Universal Robots PolyScope program: tower.urp

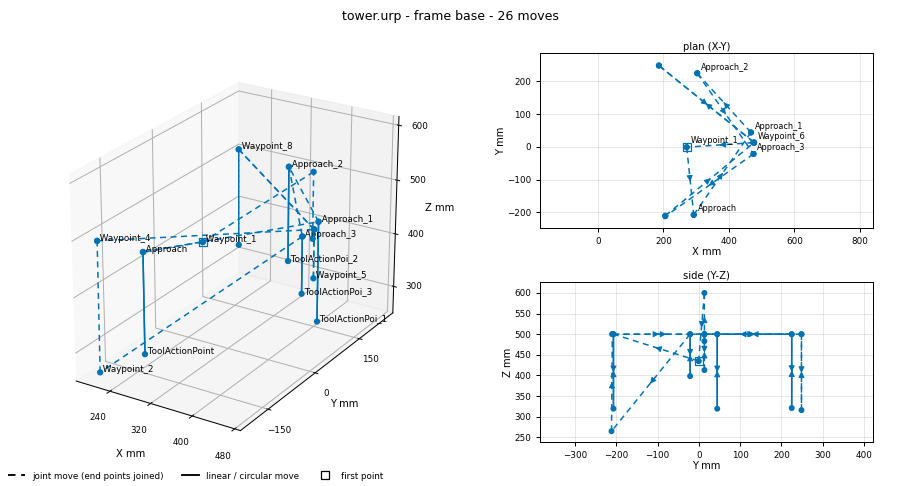
[picture p0: tool path of tower.urp in frame base, 26 of 26 moves have a stored position in this frame; points joined in program order, loops and branches not executed]
Program tower (installation=default directory=/programs createdIn=5.11.9.1010452 lastSavedIn=5.11.9.1010452 robotSerialNumber=20225200364)
Calibrated DH parameters: a=[0.00002, -0.569483, -0.54992, -0.00001, -0.000036, 0]; d=[0.180894, -146.691669, 192.918669, -46.053088, 0.119778, 0.115602]; alpha=[1.571425, -0.001534, 0.003359, 1.568739, -1.571477, 0]; deltaTheta=[0, 0.376258, -0.101074, -0.275185, -0.000002, 0]
Robot Program (runOnlyOnce=false)
  URCap RG Grip (OnRobot, OnRobot A/S) dataModel(rg-target-force=40.0, rg-target-width=0.1, Variable(key=on_return, variable(name=on_return)))
  MoveJ speed 60 deg/s, acceleration 80 deg/s^2 (useActiveTCP=true) feature=Base
    Waypoint Waypoint_1: TCP in base x=271.114 y=-0.718 z=434.853 mm, rx=2.1943 ry=2.2475 rz=0.0032 rad; joints [39.865, -70.399, -130.922, 111.401, -90.192, 38.695] deg
    Loop Counting (count=3) loopVariable(name=Loop_1)
      URCap Palletizing (polyscope-pallet-impl, Universal Robots) dataModel(palletFeature=Base, isPalletizing=true, Variable(key=name, variable(name=Pallet_1)), Variable(key=globalCountingVariable, variable(name=Pallet_1_cnt_1, initializeExpression=1)), Variable(key=layerNumberVariable, variable(name=Pallet_1_lno, initializeExpression=1)), Variable(key=layerCountingVariable, variable(name=Pallet_1_lct, initializeExpression=1)), Variable(key=handleSeparatorVariable, variable(name=Pallet_1_sep, initializeExpression=False)), Variable(key=totalCountVariable, variable(name=Pallet_1_tct, initializeExpression=1)), Variable(key=referencePoint, variable(featureName=referencePoint)), Variable(key=separatorPoint, variable(featureName=separatorPoint)), Length(key=objectHeight value=0.00001 unit=M)); state(isChildrenLocked=true)
        URCap Patterns (polyscope-pallet-impl, Universal Robots) state(isChildrenLocked=true)
          URCap Pattern (polyscope-pallet-impl, Universal Robots) dataModel(UUID=10b702ad-919e-447e-83f3-c5d126601516, patternType=LINE, objects=3, Variable(key=nameVariable, variable(name=Line_Pattern_1))); state(isChildrenLocked=true)
            URCap Item (polyscope-pallet-impl, Universal Robots) dataModel(UUID=ffec0e32-995c-4917-bab5-c4ad35439001, patternType=LINE, index=0, calibrationDeltaTheta=[-2.1094217540068572E-7, 0.37625772532806073, -0.10107441100396769, -0.2751850025766889, -1.8024952768980196E-6, 2.9402326063437956E-8], calibrationA=[2.0416891277915125E-5, -0.5694828868469309, -0.5499202125525207, -9.504674691390763E-6, -3.603723657207661E-5, 0.0], calibrationD=[0.1808937726775539, -146.69166934821124, 192.91866861971778, -46.05308757405963, 0.11977780403821288, 0.11560212559305974], calibrationAlpha=[1.5714252480212174, -0.0015337665762078037, 0.0033588312559612306, 1.5687392298942362, -1.5714772428732047, 0.0], calibrationJointChecksum=[-1490546360, -1456574554, -1506622700, -1493399207, -1492840923, -1492940558], calibrationStatus=2, calibrationValidChecksum=true, baseToFeature=[0.0, 0.0, 0.0, 0.0, 0.0, 0.0], TCPOffset=[-6.3696764394660654E-6, 1.3718254129935215E-5, 1.7975052069185704E-5, -3.893490764890671E-5, -1.8800917890220025E-5, -2.364729783574531E-6], Variable(key=variable, variable(name=StartItem_1)), JointPositions(key=jointpositions, JointPosition(key=[1], Angle(key=pos value=-0.12044 unit=RAD)), JointPosition(key=[2], Angle(key=pos value=-1.547684 unit=RAD)), JointPosition(key=[3], Angle(key=pos value=-2.267587 unit=RAD)), JointPosition(key=[4], Angle(key=pos value=2.262922 unit=RAD)), JointPosition(key=[5], Angle(key=pos value=-1.606027 unit=RAD)), JointPosition(key=[6], Angle(key=pos value=2.964753 unit=RAD))))
            URCap Item (polyscope-pallet-impl, Universal Robots) dataModel(UUID=13b54a3e-8037-4e83-825c-96e2be57fcbd, patternType=LINE, index=1, calibrationDeltaTheta=[-2.1094217540068572E-7, 0.37625772532806073, -0.10107441100396769, -0.2751850025766889, -1.8024952768980196E-6, 2.9402326063437956E-8], calibrationA=[2.0416891277915125E-5, -0.5694828868469309, -0.5499202125525207, -9.504674691390763E-6, -3.603723657207661E-5, 0.0], calibrationD=[0.1808937726775539, -146.69166934821124, 192.91866861971778, -46.05308757405963, 0.11977780403821288, 0.11560212559305974], calibrationAlpha=[1.5714252480212174, -0.0015337665762078037, 0.0033588312559612306, 1.5687392298942362, -1.5714772428732047, 0.0], calibrationJointChecksum=[-1490546360, -1456574554, -1506622700, -1493399207, -1492840923, -1492940558], calibrationStatus=2, calibrationValidChecksum=true, baseToFeature=[0.0, 0.0, 0.0, 0.0, 0.0, 0.0], TCPOffset=[1.3846566568914698E-5, -1.1531112679291633E-5, -9.126227575095847E-6, 3.8309900976807E-6, 1.563735032861701E-5, 6.604035696750426E-5], Variable(key=variable, variable(name=EndItem_1)), JointPositions(key=jointpositions, JointPosition(key=[1], Angle(key=pos value=-0.160653 unit=RAD)), JointPosition(key=[2], Angle(key=pos value=-1.420785 unit=RAD)), JointPosition(key=[3], Angle(key=pos value=-2.379964 unit=RAD)), JointPosition(key=[4], Angle(key=pos value=2.247089 unit=RAD)), JointPosition(key=[5], Angle(key=pos value=-1.606961 unit=RAD)), JointPosition(key=[6], Angle(key=pos value=2.924393 unit=RAD))))
        URCap Layers (polyscope-pallet-impl, Universal Robots) dataModel(separators=[false], selectedPatterns=[10b702ad-919e-447e-83f3-c5d126601516])
        URCap At Each Item (polyscope-pallet-impl, Universal Robots) dataModel(selectedPattern=10b702ad-919e-447e-83f3-c5d126601516, selectedPosition=ffec0e32-995c-4917-bab5-c4ad35439001, Approach_calibrationDeltaTheta=[-2.1094217540068572E-7, 0.37625772532806073, -0.10107441100396769, -0.2751850025766889, -1.8024952768980196E-6, 2.9402326063437956E-8], Approach_calibrationA=[2.0416891277915125E-5, -0.5694828868469309, -0.5499202125525207, -9.504674691390763E-6, -3.603723657207661E-5, 0.0], Approach_calibrationD=[0.1808937726775539, -146.69166934821124, 192.91866861971778, -46.05308757405963, 0.11977780403821288, 0.11560212559305974], Approach_calibrationAlpha=[1.5714252480212174, -0.0015337665762078037, 0.0033588312559612306, 1.5687392298942362, -1.5714772428732047, 0.0], Approach_calibrationJointChecksum=[-1490546360, -1456574554, -1506622700, -1493399207, -1492840923, -1492940558], Approach_calibrationStatus=2, Approach_calibrationValidChecksum=true, Approach_baseToFeature=[0.0, 0.0, 0.0, 0.0, 0.0, 0.0], Approach_TCPOffset=[4.62405650436537E-8, -1.550057465476984E-5, -1.2608941560687814E-5, -1.6491377497452102E-5, -2.0027642314724937E-5, -1.4317350537033054E-5], Exit_calibrationDeltaTheta=[-2.1094217540068572E-7, 0.37625772532806073, -0.10107441100396769, -0.2751850025766889, -1.8024952768980196E-6, 2.9402326063437956E-8], Exit_calibrationA=[2.0416891277915125E-5, -0.5694828868469309, -0.5499202125525207, -9.504674691390763E-6, -3.603723657207661E-5, 0.0], Exit_calibrationD=[0.1808937726775539, -146.69166934821124, 192.91866861971778, -46.05308757405963, 0.11977780403821288, 0.11560212559305974], Exit_calibrationAlpha=[1.5714252480212174, -0.0015337665762078037, 0.0033588312559612306, 1.5687392298942362, -1.5714772428732047, 0.0], Exit_calibrationJointChecksum=[-1490546360, -1456574554, -1506622700, -1493399207, -1492840923, -1492940558], Exit_calibrationStatus=2, Exit_calibrationValidChecksum=true, Exit_baseToFeature=[0.0, 0.0, 0.0, 0.0, 0.0, 0.0], Exit_TCPOffset=[1.1446723165831063E-5, 3.368334611741908E-5, -1.8687979546572198E-5, 3.7324910344696995E-5, 7.929792478961527E-6, 6.655834368709218E-5], currentWizardState=LANDING, Pose(key=refBaseToFeature, Position(key=posePosition, Length(key=X value=0 unit=M), Length(key=Y value=0 unit=M), Length(key=Z value=0 unit=M)), Rotation(key=poseRotation, Angle(key=RX value=0 unit=RAD), Angle(key=RY value=0 unit=RAD), Angle(key=RZ value=0 unit=RAD))), Pose(key=refPose, Position(key=posePosition, Length(key=X value=0.29256 unit=M), Length(key=Y value=-0.207279 unit=M), Length(key=Z value=0.319351 unit=M)), Rotation(key=poseRotation, Angle(key=RX value=-2.261622 unit=RAD), Angle(key=RY value=2.126603 unit=RAD), Angle(key=RZ value=0.005998 unit=RAD))), JointPositions(key=Approach_jointpositions, JointPosition(key=[1], Angle(key=pos value=-0.121062 unit=RAD)), JointPosition(key=[2], Angle(key=pos value=-1.383215 unit=RAD)), JointPosition(key=[3], Angle(key=pos value=-2.051976 unit=RAD)), JointPosition(key=[4], Angle(key=pos value=1.882818 unit=RAD)), JointPosition(key=[5], Angle(key=pos value=-1.606548 unit=RAD)), JointPosition(key=[6], Angle(key=pos value=2.962745 unit=RAD))), JointPositions(key=Exit_jointpositions, JointPosition(key=[1], Angle(key=pos value=-0.121058 unit=RAD)), JointPosition(key=[2], Angle(key=pos value=-1.383222 unit=RAD)), JointPosition(key=[3], Angle(key=pos value=-2.051981 unit=RAD)), JointPosition(key=[4], Angle(key=pos value=1.88278 unit=RAD)), JointPosition(key=[5], Angle(key=pos value=-1.606525 unit=RAD)), JointPosition(key=[6], Angle(key=pos value=2.962785 unit=RAD))))
          URCap Generated Movements (polyscope-pallet-impl, Universal Robots) state(isChildrenLocked=true)
            MoveJ speed 60 deg/s, acceleration 80 deg/s^2 (useActiveTCP=true) feature=referencePoint
              Waypoint Approach: TCP in base x=292.598 y=-207.278 z=500.013 mm, rx=-2.2616 ry=2.1265 rz=0.0059 rad; joints [-6.936, -79.254, -117.567, 107.876, -92.049, 169.752] deg; TCP offset x=0 y=0 z=0 mm, rx=0 ry=0 rz=0 rad; feature pose in base x=292.56 y=-207.279 z=319.351 mm, rx=-2.2616 ry=2.1266 rz=0.006 rad
            MoveL speed 250 mm/s, acceleration 1200 mm/s^2 (useActiveTCP=true) feature(featureName=referencePoint)
              Waypoint ToolActionPoint: TCP in base x=292.56 y=-207.279 z=319.351 mm, rx=-2.2616 ry=2.1266 rz=0.006 rad; joints [-6.9, -88.676, -129.925, 129.656, -92.019, 169.868] deg; TCP offset x=0 y=0 z=0 mm, rx=0 ry=0 rz=0 rad
            Folder Tool action
              URCap RG Grip (OnRobot, OnRobot A/S) dataModel(rg-target-force=40.0, rg-target-width=0.025)
            MoveL speed 250 mm/s, acceleration 1200 mm/s^2 (useActiveTCP=true) feature(featureName=referencePoint)
              Waypoint Exit_1: TCP in base x=292.546 y=-207.293 z=500.018 mm, rx=-2.2615 ry=2.1267 rz=0.0059 rad; joints [-6.939, -79.249, -117.57, 107.874, -92.047, 169.756] deg; TCP offset x=0 y=0 z=0 mm, rx=0 ry=0 rz=0 rad
      URCap Palletizing (polyscope-pallet-impl, Universal Robots) dataModel(palletFeature=Base, isPalletizing=true, Variable(key=name, variable(name=Pallet_2)), Variable(key=globalCountingVariable, variable(name=Pallet_2_cnt, initializeExpression=1)), Variable(key=layerNumberVariable, variable(name=Pallet_2_lno, initializeExpression=1)), Variable(key=layerCountingVariable, variable(name=Pallet_2_lct, initializeExpression=1)), Variable(key=handleSeparatorVariable, variable(name=Pallet_2_sep, initializeExpression=False)), Variable(key=totalCountVariable, variable(name=Pallet_2_tct, initializeExpression=1)), Variable(key=referencePoint, variable(featureName=referencePoin_1)), Variable(key=separatorPoint, variable(featureName=separatorPoin_1)), Length(key=objectHeight value=0.00001 unit=M)); state(isChildrenLocked=true)
        URCap Patterns (polyscope-pallet-impl, Universal Robots) state(isChildrenLocked=true)
          URCap Pattern (polyscope-pallet-impl, Universal Robots) dataModel(UUID=c8f087d8-a87e-4c62-a9c1-169a6018fd4e, patternType=LINE, objects=3, Variable(key=nameVariable, variable(name=Line_Pattern_2))); state(isChildrenLocked=true)
            URCap Item (polyscope-pallet-impl, Universal Robots) dataModel(UUID=4b9336ee-f1af-4d45-8009-66d60779b6a6, patternType=LINE, index=0, calibrationDeltaTheta=[-2.1094217540068572E-7, 0.37625772532806073, -0.10107441100396769, -0.2751850025766889, -1.8024952768980196E-6, 2.9402326063437956E-8], calibrationA=[2.0416891277915125E-5, -0.5694828868469309, -0.5499202125525207, -9.504674691390763E-6, -3.603723657207661E-5, 0.0], calibrationD=[0.1808937726775539, -146.69166934821124, 192.91866861971778, -46.05308757405963, 0.11977780403821288, 0.11560212559305974], calibrationAlpha=[1.5714252480212174, -0.0015337665762078037, 0.0033588312559612306, 1.5687392298942362, -1.5714772428732047, 0.0], calibrationJointChecksum=[-1490546360, -1456574554, -1506622700, -1493399207, -1492840923, -1492940558], calibrationStatus=2, calibrationValidChecksum=true, baseToFeature=[0.0, 0.0, 0.0, 0.0, 0.0, 0.0], TCPOffset=[4.409116630077481E-6, -1.5438319090163577E-5, -7.2719913739582864E-6, 5.112219757212625E-5, -6.20493439311258E-5, 5.425001136176107E-5], Variable(key=variable, variable(name=StartItem_2)), JointPositions(key=jointpositions, JointPosition(key=[1], Angle(key=pos value=0.474651 unit=RAD)), JointPosition(key=[2], Angle(key=pos value=-1.730821 unit=RAD)), JointPosition(key=[3], Angle(key=pos value=-2.064013 unit=RAD)), JointPosition(key=[4], Angle(key=pos value=2.256065 unit=RAD)), JointPosition(key=[5], Angle(key=pos value=-1.574508 unit=RAD)), JointPosition(key=[6], Angle(key=pos value=5.17627 unit=RAD))))
            URCap Item (polyscope-pallet-impl, Universal Robots) dataModel(UUID=a110d0e4-b9f2-4c4c-afd7-8c47bd34fb09, patternType=LINE, index=1, calibrationDeltaTheta=[-2.1094217540068572E-7, 0.37625772532806073, -0.10107441100396769, -0.2751850025766889, -1.8024952768980196E-6, 2.9402326063437956E-8], calibrationA=[2.0416891277915125E-5, -0.5694828868469309, -0.5499202125525207, -9.504674691390763E-6, -3.603723657207661E-5, 0.0], calibrationD=[0.1808937726775539, -146.69166934821124, 192.91866861971778, -46.05308757405963, 0.11977780403821288, 0.11560212559305974], calibrationAlpha=[1.5714252480212174, -0.0015337665762078037, 0.0033588312559612306, 1.5687392298942362, -1.5714772428732047, 0.0], calibrationJointChecksum=[-1490546360, -1456574554, -1506622700, -1493399207, -1492840923, -1492940558], calibrationStatus=2, calibrationValidChecksum=true, baseToFeature=[0.0, 0.0, 0.0, 0.0, 0.0, 0.0], TCPOffset=[-1.4380333733965411E-5, -5.264472437292028E-6, -9.358425566097228E-6, -1.0911522351191877E-5, -4.3963888238967464E-5, 2.2254276518748705E-5], Variable(key=variable, variable(name=EndItem_2)), JointPositions(key=jointpositions, JointPosition(key=[1], Angle(key=pos value=0.326248 unit=RAD)), JointPosition(key=[2], Angle(key=pos value=-1.729038 unit=RAD)), JointPosition(key=[3], Angle(key=pos value=-2.066304 unit=RAD)), JointPosition(key=[4], Angle(key=pos value=2.256092 unit=RAD)), JointPosition(key=[5], Angle(key=pos value=-1.579334 unit=RAD)), JointPosition(key=[6], Angle(key=pos value=5.027941 unit=RAD))))
        URCap Layers (polyscope-pallet-impl, Universal Robots) dataModel(separators=[false], selectedPatterns=[c8f087d8-a87e-4c62-a9c1-169a6018fd4e])
        URCap At Each Item (polyscope-pallet-impl, Universal Robots) dataModel(selectedPattern=c8f087d8-a87e-4c62-a9c1-169a6018fd4e, selectedPosition=4b9336ee-f1af-4d45-8009-66d60779b6a6, Approach_calibrationDeltaTheta=[-2.1094217540068572E-7, 0.37625772532806073, -0.10107441100396769, -0.2751850025766889, -1.8024952768980196E-6, 2.9402326063437956E-8], Approach_calibrationA=[2.0416891277915125E-5, -0.5694828868469309, -0.5499202125525207, -9.504674691390763E-6, -3.603723657207661E-5, 0.0], Approach_calibrationD=[0.1808937726775539, -146.69166934821124, 192.91866861971778, -46.05308757405963, 0.11977780403821288, 0.11560212559305974], Approach_calibrationAlpha=[1.5714252480212174, -0.0015337665762078037, 0.0033588312559612306, 1.5687392298942362, -1.5714772428732047, 0.0], Approach_calibrationJointChecksum=[-1490546360, -1456574554, -1506622700, -1493399207, -1492840923, -1492940558], Approach_calibrationStatus=2, Approach_calibrationValidChecksum=true, Approach_baseToFeature=[0.0, 0.0, 0.0, 0.0, 0.0, 0.0], Approach_TCPOffset=[1.1639698013432564E-5, -8.846874539378269E-6, 1.1133412487873695E-5, 1.6117839583191827E-5, 5.374636367245953E-5, 1.074239401068827E-6], Exit_calibrationDeltaTheta=[-2.1094217540068572E-7, 0.37625772532806073, -0.10107441100396769, -0.2751850025766889, -1.8024952768980196E-6, 2.9402326063437956E-8], Exit_calibrationA=[2.0416891277915125E-5, -0.5694828868469309, -0.5499202125525207, -9.504674691390763E-6, -3.603723657207661E-5, 0.0], Exit_calibrationD=[0.1808937726775539, -146.69166934821124, 192.91866861971778, -46.05308757405963, 0.11977780403821288, 0.11560212559305974], Exit_calibrationAlpha=[1.5714252480212174, -0.0015337665762078037, 0.0033588312559612306, 1.5687392298942362, -1.5714772428732047, 0.0], Exit_calibrationJointChecksum=[-1490546360, -1456574554, -1506622700, -1493399207, -1492840923, -1492940558], Exit_calibrationStatus=2, Exit_calibrationValidChecksum=true, Exit_baseToFeature=[0.0, 0.0, 0.0, 0.0, 0.0, 0.0], Exit_TCPOffset=[-6.688063342030759E-8, 1.0405827377074628E-5, -5.466452467406402E-6, 3.1866222240658605E-5, 4.424926447771402E-5, -4.5818155317012656E-5], currentWizardState=LANDING, Pose(key=refBaseToFeature, Position(key=posePosition, Length(key=X value=0 unit=M), Length(key=Y value=0 unit=M), Length(key=Z value=0 unit=M)), Rotation(key=poseRotation, Angle(key=RX value=0 unit=RAD), Angle(key=RY value=0 unit=RAD), Angle(key=RZ value=0 unit=RAD))), Pose(key=refPose, Position(key=posePosition, Length(key=X value=0.46728 unit=M), Length(key=Y value=0.044349 unit=M), Length(key=Z value=0.319231 unit=M)), Rotation(key=poseRotation, Angle(key=RX value=-0.0243 unit=RAD), Angle(key=RY value=3.112588 unit=RAD), Angle(key=RZ value=0.024192 unit=RAD))), JointPositions(key=Approach_jointpositions, JointPosition(key=[1], Angle(key=pos value=0.474285 unit=RAD)), JointPosition(key=[2], Angle(key=pos value=-1.582914 unit=RAD)), JointPosition(key=[3], Angle(key=pos value=-1.86876 unit=RAD)), JointPosition(key=[4], Angle(key=pos value=1.91298 unit=RAD)), JointPosition(key=[5], Angle(key=pos value=-1.574975 unit=RAD)), JointPosition(key=[6], Angle(key=pos value=5.174807 unit=RAD))), JointPositions(key=Exit_jointpositions, JointPosition(key=[1], Angle(key=pos value=0.474302 unit=RAD)), JointPosition(key=[2], Angle(key=pos value=-1.582917 unit=RAD)), JointPosition(key=[3], Angle(key=pos value=-1.868746 unit=RAD)), JointPosition(key=[4], Angle(key=pos value=1.913021 unit=RAD)), JointPosition(key=[5], Angle(key=pos value=-1.574942 unit=RAD)), JointPosition(key=[6], Angle(key=pos value=5.174836 unit=RAD))))
          URCap Generated Movements (polyscope-pallet-impl, Universal Robots) state(isChildrenLocked=true)
            MoveJ speed 60 deg/s, acceleration 80 deg/s^2 (useActiveTCP=true) feature=referencePoin_1
              Waypoint Approach_1: TCP in base x=467.265 y=44.333 z=499.988 mm, rx=-0.0243 ry=3.1126 rz=0.0243 rad; joints [27.174, -90.694, -107.074, 109.604, -90.24, 296.494] deg; TCP offset x=0 y=0 z=0 mm, rx=0 ry=0 rz=0 rad; feature pose in base x=467.28 y=44.349 z=319.231 mm, rx=-0.0243 ry=3.1126 rz=0.0242 rad
            MoveL speed 250 mm/s, acceleration 1200 mm/s^2 (useActiveTCP=true) feature(featureName=referencePoin_1)
              Waypoint ToolActionPoi_1: TCP in base x=467.28 y=44.349 z=319.231 mm, rx=-0.0243 ry=3.1126 rz=0.0242 rad; joints [27.195, -99.167, -118.26, 129.264, -90.208, 296.581] deg; TCP offset x=0 y=0 z=0 mm, rx=0 ry=0 rz=0 rad
            Folder Tool action
              URCap RG Grip (OnRobot, OnRobot A/S) dataModel(rg-target-force=40.0, rg-target-width=0.03)
            MoveL speed 250 mm/s, acceleration 1200 mm/s^2 (useActiveTCP=true) feature(featureName=referencePoin_1)
              Waypoint Exit_2: TCP in base x=467.286 y=44.361 z=500.006 mm, rx=-0.0243 ry=3.1125 rz=0.0242 rad; joints [27.177, -90.695, -107.071, 109.605, -90.237, 296.495] deg; TCP offset x=0 y=0 z=0 mm, rx=0 ry=0 rz=0 rad
    Loop Counting (count=3) loopVariable(name=Loop_2)
      URCap Palletizing (polyscope-pallet-impl, Universal Robots) dataModel(palletFeature=Base, isPalletizing=true, Variable(key=name, variable(name=Pallet_3)), Variable(key=globalCountingVariable, variable(name=Pallet_3_cnt, initializeExpression=1)), Variable(key=layerNumberVariable, variable(name=Pallet_3_lno, initializeExpression=1)), Variable(key=layerCountingVariable, variable(name=Pallet_3_lct, initializeExpression=1)), Variable(key=handleSeparatorVariable, variable(name=Pallet_3_sep, initializeExpression=False)), Variable(key=totalCountVariable, variable(name=Pallet_3_tct, initializeExpression=1)), Variable(key=referencePoint, variable(featureName=referencePoin_2)), Variable(key=separatorPoint, variable(featureName=separatorPoin_2)), Length(key=objectHeight value=0.00001 unit=M)); state(isChildrenLocked=true)
        URCap Patterns (polyscope-pallet-impl, Universal Robots) state(isChildrenLocked=true)
          URCap Pattern (polyscope-pallet-impl, Universal Robots) dataModel(UUID=69e63fbd-ac57-40a8-8514-40e488ea7127, patternType=LINE, objects=3, Variable(key=nameVariable, variable(name=Line_Pattern_3))); state(isChildrenLocked=true)
            URCap Item (polyscope-pallet-impl, Universal Robots) dataModel(UUID=d74f1e55-d7a4-4b92-9c14-17e5686717f3, patternType=LINE, index=0, calibrationDeltaTheta=[-2.1094217540068572E-7, 0.37625772532806073, -0.10107441100396769, -0.2751850025766889, -1.8024952768980196E-6, 2.9402326063437956E-8], calibrationA=[2.0416891277915125E-5, -0.5694828868469309, -0.5499202125525207, -9.504674691390763E-6, -3.603723657207661E-5, 0.0], calibrationD=[0.1808937726775539, -146.69166934821124, 192.91866861971778, -46.05308757405963, 0.11977780403821288, 0.11560212559305974], calibrationAlpha=[1.5714252480212174, -0.0015337665762078037, 0.0033588312559612306, 1.5687392298942362, -1.5714772428732047, 0.0], calibrationJointChecksum=[-1490546360, -1456574554, -1506622700, -1493399207, -1492840923, -1492940558], calibrationStatus=2, calibrationValidChecksum=true, baseToFeature=[0.0, 0.0, 0.0, 0.0, 0.0, 0.0], TCPOffset=[1.2985872193088666E-5, -6.705328385370191E-6, -7.116337871981848E-6, 1.0691414030932002E-5, -1.1363978627081674E-5, -2.520531805839135E-5], Variable(key=variable, variable(name=StartItem_3)), JointPositions(key=jointpositions, JointPosition(key=[1], Angle(key=pos value=1.118695 unit=RAD)), JointPosition(key=[2], Angle(key=pos value=-1.583327 unit=RAD)), JointPosition(key=[3], Angle(key=pos value=-2.233039 unit=RAD)), JointPosition(key=[4], Angle(key=pos value=2.246663 unit=RAD)), JointPosition(key=[5], Angle(key=pos value=-1.572601 unit=RAD)), JointPosition(key=[6], Angle(key=pos value=1.099535 unit=RAD))))
            URCap Item (polyscope-pallet-impl, Universal Robots) dataModel(UUID=ef41c16a-ce02-4892-a50c-4f21fb1603f3, patternType=LINE, index=1, calibrationDeltaTheta=[-2.1094217540068572E-7, 0.37625772532806073, -0.10107441100396769, -0.2751850025766889, -1.8024952768980196E-6, 2.9402326063437956E-8], calibrationA=[2.0416891277915125E-5, -0.5694828868469309, -0.5499202125525207, -9.504674691390763E-6, -3.603723657207661E-5, 0.0], calibrationD=[0.1808937726775539, -146.69166934821124, 192.91866861971778, -46.05308757405963, 0.11977780403821288, 0.11560212559305974], calibrationAlpha=[1.5714252480212174, -0.0015337665762078037, 0.0033588312559612306, 1.5687392298942362, -1.5714772428732047, 0.0], calibrationJointChecksum=[-1490546360, -1456574554, -1506622700, -1493399207, -1492840923, -1492940558], calibrationStatus=2, calibrationValidChecksum=true, baseToFeature=[0.0, 0.0, 0.0, 0.0, 0.0, 0.0], TCPOffset=[-5.307224317796511E-7, -5.42229024316776E-6, -2.5424014468145018E-6, -2.8661002424582808E-5, -9.543783619449082E-6, -3.3871828536279686E-5], Variable(key=variable, variable(name=EndItem_3)), JointPositions(key=jointpositions, JointPosition(key=[1], Angle(key=pos value=1.374483 unit=RAD)), JointPosition(key=[2], Angle(key=pos value=-1.463304 unit=RAD)), JointPosition(key=[3], Angle(key=pos value=-2.345439 unit=RAD)), JointPosition(key=[4], Angle(key=pos value=2.238646 unit=RAD)), JointPosition(key=[5], Angle(key=pos value=-1.572398 unit=RAD)), JointPosition(key=[6], Angle(key=pos value=1.355219 unit=RAD))))
        URCap Layers (polyscope-pallet-impl, Universal Robots) dataModel(separators=[false], selectedPatterns=[69e63fbd-ac57-40a8-8514-40e488ea7127])
        URCap At Each Item (polyscope-pallet-impl, Universal Robots) dataModel(selectedPattern=69e63fbd-ac57-40a8-8514-40e488ea7127, selectedPosition=d74f1e55-d7a4-4b92-9c14-17e5686717f3, Approach_calibrationDeltaTheta=[-2.1094217540068572E-7, 0.37625772532806073, -0.10107441100396769, -0.2751850025766889, -1.8024952768980196E-6, 2.9402326063437956E-8], Approach_calibrationA=[2.0416891277915125E-5, -0.5694828868469309, -0.5499202125525207, -9.504674691390763E-6, -3.603723657207661E-5, 0.0], Approach_calibrationD=[0.1808937726775539, -146.69166934821124, 192.91866861971778, -46.05308757405963, 0.11977780403821288, 0.11560212559305974], Approach_calibrationAlpha=[1.5714252480212174, -0.0015337665762078037, 0.0033588312559612306, 1.5687392298942362, -1.5714772428732047, 0.0], Approach_calibrationJointChecksum=[-1490546360, -1456574554, -1506622700, -1493399207, -1492840923, -1492940558], Approach_calibrationStatus=2, Approach_calibrationValidChecksum=true, Approach_baseToFeature=[0.0, 0.0, 0.0, 0.0, 0.0, 0.0], Approach_TCPOffset=[-3.973529929257591E-7, 1.169112545090778E-5, 7.133541923498576E-6, -2.6345289464818864E-5, -4.662160305502815E-5, -1.1711297164837408E-5], Exit_calibrationDeltaTheta=[-2.1094217540068572E-7, 0.37625772532806073, -0.10107441100396769, -0.2751850025766889, -1.8024952768980196E-6, 2.9402326063437956E-8], Exit_calibrationA=[2.0416891277915125E-5, -0.5694828868469309, -0.5499202125525207, -9.504674691390763E-6, -3.603723657207661E-5, 0.0], Exit_calibrationD=[0.1808937726775539, -146.69166934821124, 192.91866861971778, -46.05308757405963, 0.11977780403821288, 0.11560212559305974], Exit_calibrationAlpha=[1.5714252480212174, -0.0015337665762078037, 0.0033588312559612306, 1.5687392298942362, -1.5714772428732047, 0.0], Exit_calibrationJointChecksum=[-1490546360, -1456574554, -1506622700, -1493399207, -1492840923, -1492940558], Exit_calibrationStatus=2, Exit_calibrationValidChecksum=true, Exit_baseToFeature=[0.0, 0.0, 0.0, 0.0, 0.0, 0.0], Exit_TCPOffset=[8.652881060000617E-7, 5.1828311730117704E-6, 2.66209812420648E-5, 5.491666351403043E-6, -3.31371066403185E-5, 2.701581242020385E-5], currentWizardState=SHOW_DONE, Pose(key=refBaseToFeature, Position(key=posePosition, Length(key=X value=0 unit=M), Length(key=Y value=0 unit=M), Length(key=Z value=0 unit=M)), Rotation(key=poseRotation, Angle(key=RX value=0 unit=RAD), Angle(key=RY value=0 unit=RAD), Angle(key=RZ value=0 unit=RAD))), Pose(key=refPose, Position(key=posePosition, Length(key=X value=0.303191 unit=M), Length(key=Y value=0.224938 unit=M), Length(key=Z value=0.320986 unit=M)), Rotation(key=poseRotation, Angle(key=RX value=2.194265 unit=RAD), Angle(key=RY value=2.24748 unit=RAD), Angle(key=RZ value=0.003234 unit=RAD))), JointPositions(key=Approach_jointpositions, JointPosition(key=[1], Angle(key=pos value=1.118094 unit=RAD)), JointPosition(key=[2], Angle(key=pos value=-1.421731 unit=RAD)), JointPosition(key=[3], Angle(key=pos value=-2.024324 unit=RAD)), JointPosition(key=[4], Angle(key=pos value=1.876398 unit=RAD)), JointPosition(key=[5], Angle(key=pos value=-1.573128 unit=RAD)), JointPosition(key=[6], Angle(key=pos value=1.09767 unit=RAD))), JointPositions(key=Exit_jointpositions, JointPosition(key=[1], Angle(key=pos value=1.118152 unit=RAD)), JointPosition(key=[2], Angle(key=pos value=-1.42171 unit=RAD)), JointPosition(key=[3], Angle(key=pos value=-2.024361 unit=RAD)), JointPosition(key=[4], Angle(key=pos value=1.876324 unit=RAD)), JointPosition(key=[5], Angle(key=pos value=-1.573107 unit=RAD)), JointPosition(key=[6], Angle(key=pos value=1.097669 unit=RAD))))
          URCap Generated Movements (polyscope-pallet-impl, Universal Robots) state(isChildrenLocked=true)
            MoveJ speed 60 deg/s, acceleration 80 deg/s^2 (useActiveTCP=true) feature=referencePoin_2
              Waypoint Approach_2: TCP in base x=303.211 y=224.943 z=499.993 mm, rx=2.1943 ry=2.2474 rz=0.0033 rad; joints [64.061, -81.461, -115.985, 107.509, -90.131, 62.89] deg; TCP offset x=0 y=0 z=0 mm, rx=0 ry=0 rz=0 rad; feature pose in base x=303.191 y=224.938 z=320.986 mm, rx=2.1943 ry=2.2475 rz=0.0032 rad
            MoveL speed 250 mm/s, acceleration 1200 mm/s^2 (useActiveTCP=true) feature(featureName=referencePoin_2)
              Waypoint ToolActionPoi_2: TCP in base x=303.191 y=224.938 z=320.986 mm, rx=2.1943 ry=2.2475 rz=0.0032 rad; joints [64.096, -90.718, -127.944, 128.724, -90.103, 62.999] deg; TCP offset x=0 y=0 z=0 mm, rx=0 ry=0 rz=0 rad
            Folder Tool action
              URCap RG Grip (OnRobot, OnRobot A/S) dataModel(rg-target-force=40.0, rg-target-width=0.025)
            MoveL speed 250 mm/s, acceleration 1200 mm/s^2 (useActiveTCP=true) feature(featureName=referencePoin_2)
              Waypoint Exit_3: TCP in base x=303.182 y=224.937 z=499.973 mm, rx=2.1943 ry=2.2474 rz=0.0031 rad; joints [64.065, -81.46, -115.989, 107.507, -90.132, 62.893] deg; TCP offset x=0 y=0 z=0 mm, rx=0 ry=0 rz=0 rad
      URCap Palletizing (polyscope-pallet-impl, Universal Robots) dataModel(palletFeature=Base, isPalletizing=true, Variable(key=name, variable(name=Pallet_4)), Variable(key=globalCountingVariable, variable(name=Pallet_4_cnt, initializeExpression=1)), Variable(key=layerNumberVariable, variable(name=Pallet_4_lno, initializeExpression=1)), Variable(key=layerCountingVariable, variable(name=Pallet_4_lct, initializeExpression=1)), Variable(key=handleSeparatorVariable, variable(name=Pallet_4_sep, initializeExpression=False)), Variable(key=totalCountVariable, variable(name=Pallet_4_tct, initializeExpression=1)), Variable(key=referencePoint, variable(featureName=referencePoin_3)), Variable(key=separatorPoint, variable(featureName=separatorPoin_3)), Length(key=objectHeight value=0.00001 unit=M)); state(isChildrenLocked=true)
        URCap Patterns (polyscope-pallet-impl, Universal Robots) state(isChildrenLocked=true)
          URCap Pattern (polyscope-pallet-impl, Universal Robots) dataModel(UUID=02354257-159c-4745-9de3-4e64df3cce66, patternType=LINE, objects=3, Variable(key=nameVariable, variable(name=Line_Pattern_4))); state(isChildrenLocked=true)
            URCap Item (polyscope-pallet-impl, Universal Robots) dataModel(UUID=2191eea5-a3bf-41bd-8f05-986646ba22a6, patternType=LINE, index=0, calibrationDeltaTheta=[-2.1094217540068572E-7, 0.37625772532806073, -0.10107441100396769, -0.2751850025766889, -1.8024952768980196E-6, 2.9402326063437956E-8], calibrationA=[2.0416891277915125E-5, -0.5694828868469309, -0.5499202125525207, -9.504674691390763E-6, -3.603723657207661E-5, 0.0], calibrationD=[0.1808937726775539, -146.69166934821124, 192.91866861971778, -46.05308757405963, 0.11977780403821288, 0.11560212559305974], calibrationAlpha=[1.5714252480212174, -0.0015337665762078037, 0.0033588312559612306, 1.5687392298942362, -1.5714772428732047, 0.0], calibrationJointChecksum=[-1490546360, -1456574554, -1506622700, -1493399207, -1492840923, -1492940558], calibrationStatus=2, calibrationValidChecksum=true, baseToFeature=[0.0, 0.0, 0.0, 0.0, 0.0, 0.0], TCPOffset=[2.1473476097266797E-7, -1.0619135056781637E-5, -1.684877696334075E-5, 2.9450928766290354E-5, 2.4808781527186736E-7, 2.0484144679390314E-5], Variable(key=variable, variable(name=StartItem_4)), JointPositions(key=jointpositions, JointPosition(key=[1], Angle(key=pos value=0.331823 unit=RAD)), JointPosition(key=[2], Angle(key=pos value=-1.667002 unit=RAD)), JointPosition(key=[3], Angle(key=pos value=-1.980696 unit=RAD)), JointPosition(key=[4], Angle(key=pos value=2.075957 unit=RAD)), JointPosition(key=[5], Angle(key=pos value=-1.575935 unit=RAD)), JointPosition(key=[6], Angle(key=pos value=-1.251483 unit=RAD))))
            URCap Item (polyscope-pallet-impl, Universal Robots) dataModel(UUID=a4ccdb19-ac43-48e7-abc6-d9b3ebcec3d8, patternType=LINE, index=1, calibrationDeltaTheta=[-2.1094217540068572E-7, 0.37625772532806073, -0.10107441100396769, -0.2751850025766889, -1.8024952768980196E-6, 2.9402326063437956E-8], calibrationA=[2.0416891277915125E-5, -0.5694828868469309, -0.5499202125525207, -9.504674691390763E-6, -3.603723657207661E-5, 0.0], calibrationD=[0.1808937726775539, -146.69166934821124, 192.91866861971778, -46.05308757405963, 0.11977780403821288, 0.11560212559305974], calibrationAlpha=[1.5714252480212174, -0.0015337665762078037, 0.0033588312559612306, 1.5687392298942362, -1.5714772428732047, 0.0], calibrationJointChecksum=[-1490546360, -1456574554, -1506622700, -1493399207, -1492840923, -1492940558], calibrationStatus=2, calibrationValidChecksum=true, baseToFeature=[0.0, 0.0, 0.0, 0.0, 0.0, 0.0], TCPOffset=[-6.467086302586189E-6, -3.802894154303349E-6, 3.230648946939141E-5, -7.782766569128539E-6, 6.097839921019588E-5, 5.012173512466323E-5], Variable(key=variable, variable(name=EndItem_4)), JointPositions(key=jointpositions, JointPosition(key=[1], Angle(key=pos value=0.474834 unit=RAD)), JointPosition(key=[2], Angle(key=pos value=-1.675955 unit=RAD)), JointPosition(key=[3], Angle(key=pos value=-1.97092 unit=RAD)), JointPosition(key=[4], Angle(key=pos value=2.075325 unit=RAD)), JointPosition(key=[5], Angle(key=pos value=-1.575982 unit=RAD)), JointPosition(key=[6], Angle(key=pos value=-1.108497 unit=RAD))))
        URCap Layers (polyscope-pallet-impl, Universal Robots) dataModel(separators=[false], selectedPatterns=[02354257-159c-4745-9de3-4e64df3cce66])
        URCap At Each Item (polyscope-pallet-impl, Universal Robots) dataModel(selectedPattern=02354257-159c-4745-9de3-4e64df3cce66, selectedPosition=2191eea5-a3bf-41bd-8f05-986646ba22a6, Approach_calibrationDeltaTheta=[-2.1094217540068572E-7, 0.37625772532806073, -0.10107441100396769, -0.2751850025766889, -1.8024952768980196E-6, 2.9402326063437956E-8], Approach_calibrationA=[2.0416891277915125E-5, -0.5694828868469309, -0.5499202125525207, -9.504674691390763E-6, -3.603723657207661E-5, 0.0], Approach_calibrationD=[0.1808937726775539, -146.69166934821124, 192.91866861971778, -46.05308757405963, 0.11977780403821288, 0.11560212559305974], Approach_calibrationAlpha=[1.5714252480212174, -0.0015337665762078037, 0.0033588312559612306, 1.5687392298942362, -1.5714772428732047, 0.0], Approach_calibrationJointChecksum=[-1490546360, -1456574554, -1506622700, -1493399207, -1492840923, -1492940558], Approach_calibrationStatus=2, Approach_calibrationValidChecksum=true, Approach_baseToFeature=[0.0, 0.0, 0.0, 0.0, 0.0, 0.0], Approach_TCPOffset=[-4.8549868723046785E-6, -1.343598116847547E-5, -4.4727514389997225E-6, 7.711808721261738E-6, -1.8311670577592164E-5, 1.549552527328898E-5], Exit_calibrationDeltaTheta=[-2.1094217540068572E-7, 0.37625772532806073, -0.10107441100396769, -0.2751850025766889, -1.8024952768980196E-6, 2.9402326063437956E-8], Exit_calibrationA=[2.0416891277915125E-5, -0.5694828868469309, -0.5499202125525207, -9.504674691390763E-6, -3.603723657207661E-5, 0.0], Exit_calibrationD=[0.1808937726775539, -146.69166934821124, 192.91866861971778, -46.05308757405963, 0.11977780403821288, 0.11560212559305974], Exit_calibrationAlpha=[1.5714252480212174, -0.0015337665762078037, 0.0033588312559612306, 1.5687392298942362, -1.5714772428732047, 0.0], Exit_calibrationJointChecksum=[-1490546360, -1456574554, -1506622700, -1493399207, -1492840923, -1492940558], Exit_calibrationStatus=2, Exit_calibrationValidChecksum=true, Exit_baseToFeature=[0.0, 0.0, 0.0, 0.0, 0.0, 0.0], Exit_TCPOffset=[7.417940817655566E-6, -1.1578098806756115E-5, -8.794698510783405E-6, 5.938538054833778E-5, -5.6794407952116924E-5, 1.3661997192754913E-5], currentWizardState=SHOW_DONE, Pose(key=refBaseToFeature, Position(key=posePosition, Length(key=X value=0 unit=M), Length(key=Y value=0 unit=M), Length(key=Z value=0 unit=M)), Rotation(key=poseRotation, Angle(key=RX value=0 unit=RAD), Angle(key=RY value=0 unit=RAD), Angle(key=RZ value=0 unit=RAD))), Pose(key=refPose, Position(key=posePosition, Length(key=X value=0.475201 unit=M), Length(key=Y value=-0.021335 unit=M), Length(key=Z value=0.398423 unit=M)), Rotation(key=poseRotation, Angle(key=RX value=0.026388 unit=RAD), Angle(key=RY value=-3.140553 unit=RAD), Angle(key=RZ value=-0.002951 unit=RAD))), JointPositions(key=Approach_jointpositions, JointPosition(key=[1], Angle(key=pos value=0.3292 unit=RAD)), JointPosition(key=[2], Angle(key=pos value=-1.602345 unit=RAD)), JointPosition(key=[3], Angle(key=pos value=-1.856028 unit=RAD)), JointPosition(key=[4], Angle(key=pos value=1.886544 unit=RAD)), JointPosition(key=[5], Angle(key=pos value=-1.576153 unit=RAD)), JointPosition(key=[6], Angle(key=pos value=-1.254782 unit=RAD))), JointPositions(key=Exit_jointpositions, JointPosition(key=[1], Angle(key=pos value=0.329193 unit=RAD)), JointPosition(key=[2], Angle(key=pos value=-1.602406 unit=RAD)), JointPosition(key=[3], Angle(key=pos value=-1.855942 unit=RAD)), JointPosition(key=[4], Angle(key=pos value=1.886622 unit=RAD)), JointPosition(key=[5], Angle(key=pos value=-1.5761 unit=RAD)), JointPosition(key=[6], Angle(key=pos value=-1.254773 unit=RAD))))
          URCap Generated Movements (polyscope-pallet-impl, Universal Robots) state(isChildrenLocked=true)
            MoveJ speed 60 deg/s, acceleration 80 deg/s^2 (useActiveTCP=true) feature=referencePoin_3
              Waypoint Approach_3: TCP in base x=475.196 y=-21.344 z=500.004 mm, rx=0.0264 ry=-3.1405 rz=-0.003 rad; joints [18.86, -91.808, -106.342, 108.091, -90.306, -71.894] deg; TCP offset x=0 y=0 z=0 mm, rx=0 ry=0 rz=0 rad; feature pose in base x=475.201 y=-21.335 z=398.423 mm, rx=0.0264 ry=-3.1406 rz=-0.003 rad
            MoveL speed 250 mm/s, acceleration 1200 mm/s^2 (useActiveTCP=true) feature(featureName=referencePoin_3)
              Waypoint ToolActionPoi_3: TCP in base x=475.201 y=-21.335 z=398.423 mm, rx=0.0264 ry=-3.1406 rz=-0.003 rad; joints [18.872, -95.829, -113.131, 118.905, -90.294, -71.845] deg; TCP offset x=0 y=0 z=0 mm, rx=0 ry=0 rz=0 rad
            Folder Tool action
              URCap RG Grip (OnRobot, OnRobot A/S) dataModel(rg-target-force=40.0, rg-target-width=0.03)
            MoveL speed 250 mm/s, acceleration 1200 mm/s^2 (useActiveTCP=true) feature(featureName=referencePoin_3)
              Waypoint Exit_4: TCP in base x=475.236 y=-21.334 z=500.009 mm, rx=0.0264 ry=-3.1406 rz=-0.0028 rad; joints [18.861, -91.809, -106.338, 108.096, -90.3, -71.892] deg; TCP offset x=0 y=0 z=0 mm, rx=0 ry=0 rz=0 rad
    URCap RG Grip (OnRobot, OnRobot A/S) dataModel(rg-target-force=40.0, rg-target-width=0.1)
    Waypoint Waypoint_2: TCP in base x=205.755 y=-211.952 z=264.758 mm, rx=2.1944 ry=2.2474 rz=0.0032 rad; joints [-9.68, -86.405, -139.741, 136.198, -90.245, -10.753] deg
    URCap RG Grip (OnRobot, OnRobot A/S) dataModel(rg-target-force=40.0, rg-target-width=0.075)
    Waypoint Waypoint_4: TCP in base x=205.807 y=-210.051 z=500.009 mm, rx=2.1941 ry=2.2475 rz=0.003 rad; joints [-9.295, -71.324, -123.469, 104.849, -90.281, -10.493] deg
    URCap RG Grip (OnRobot, OnRobot A/S) dataModel(rg-target-force=40.0, rg-target-width=0.075)
    Waypoint Waypoint_4: TCP in base x=205.807 y=-210.051 z=500.009 mm, rx=2.1941 ry=2.2475 rz=0.003 rad; joints [-9.295, -71.324, -123.469, 104.849, -90.281, -10.493] deg
    Waypoint Waypoint_6: TCP in base x=477.044 y=13.254 z=499.999 mm, rx=2.2155 ry=2.2236 rz=-0.0002 rad; joints [23.018, -91.926, -106.205, 108.141, -90.044, 23.018] deg
    Waypoint Waypoint_5: TCP in base x=477.046 y=13.273 z=412.952 mm, rx=2.2156 ry=2.2237 rz=-0.0002 rad; joints [23.029, -95.249, -112.112, 117.369, -90.038, 23.061] deg
    URCap RG Grip (OnRobot, OnRobot A/S) dataModel(rg-target-force=40.0, rg-target-width=0.1)
    Waypoint Waypoint_6: TCP in base x=477.044 y=13.254 z=499.999 mm, rx=2.2155 ry=2.2236 rz=-0.0002 rad; joints [23.018, -91.926, -106.205, 108.141, -90.044, 23.018] deg
    Waypoint Waypoint_8: TCP in base x=186.058 y=248.584 z=499.987 mm, rx=2.2156 ry=2.2236 rz=-0.0003 rad; joints [87.353, -73.514, -122.059, 105.426, -90.11, 87.331] deg
    Waypoint Waypoint_7: TCP in base x=186.053 y=248.622 z=315.838 mm, rx=2.2156 ry=2.2237 rz=-0.0002 rad; joints [87.408, -83.581, -135.314, 128.753, -90.08, 87.47] deg
    URCap RG Grip (OnRobot, OnRobot A/S) dataModel(rg-target-force=40.0, rg-target-width=0.025)
    Waypoint Waypoint_8: TCP in base x=186.058 y=248.584 z=499.987 mm, rx=2.2156 ry=2.2236 rz=-0.0003 rad; joints [87.353, -73.514, -122.059, 105.426, -90.11, 87.331] deg
    Waypoint Waypoint_6: TCP in base x=477.044 y=13.254 z=499.999 mm, rx=2.2155 ry=2.2236 rz=-0.0002 rad; joints [23.018, -91.926, -106.205, 108.141, -90.044, 23.018] deg
    Waypoint Waypoint_9: TCP in base x=474.536 y=13.241 z=482.99 mm, rx=2.2155 ry=2.2236 rz=-0.0002 rad; joints [23.146, -92.217, -107.706, 109.933, -90.042, 23.152] deg
    URCap RG Grip (OnRobot, OnRobot A/S) dataModel(rg-target-force=40.0, rg-target-width=0.03)
    Waypoint Waypoint_10: TCP in base x=474.544 y=13.277 z=599.981 mm, rx=2.2155 ry=2.2237 rz=-0.0002 rad; joints [23.138, -89.535, -98.327, 97.873, -90.046, 23.1] deg
    Waypoint Waypoint_1: TCP in base x=271.114 y=-0.718 z=434.853 mm, rx=2.1943 ry=2.2475 rz=0.0032 rad; joints [39.865, -70.399, -130.922, 111.401, -90.192, 38.695] deg
    Halt
